FUNCTION_BLOCK L1_Merge2Cmd (* Basic Function Block Type *)
  (* Standard: 61499-2 *)
  (* Version 0.0, 2015-03-18, EQUEROL, UJI *)
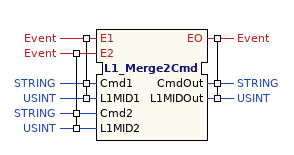
  EVENT_INPUT
    E1 WITH Cmd1, L1MID1; (* Event to merge 1 *)
    E2 WITH Cmd2, L1MID2; (* Event to merge 2 *)
  END_EVENT
  EVENT_OUTPUT
    EO WITH CmdOut, L1MIDOut; (* Initialization Confirm *)
  END_EVENT
  VAR_INPUT
    Cmd1 : STRING; (* Command with event 1 *)
    L1MID1 : USINT; (* Layer 1 multicast ID with 1 *)
    Cmd2 : STRING; (* Command with event 2 *)
    L1MID2 : USINT; (* Layer 1 multicast ID with 2 *)
  END_VAR
  VAR_OUTPUT
    CmdOut : STRING; (* Command out *)
    L1MIDOut : USINT; (* Layer 1 multicast ID *)
  END_VAR
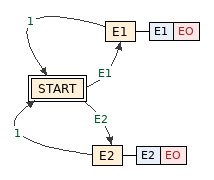
  EC_STATES
    START; (* Initial State *)
    E1 : E1 -> EO; (* Initialization *)
    E2 : E2 -> EO; (* Normal execution *)
  END_STATES
  EC_TRANSITIONS
    START TO E1 := E1;
    E1 TO START := 1;
    START TO E2 := E2;
    E2 TO START := 1;
  END_TRANSITIONS
  ALGORITHM E1 IN ST: (* Event 1 algo *)
CmdOut := Cmd1;
L1MIDOut := L1MID1;
  END_ALGORITHM
  ALGORITHM E2 IN ST: (* Event 2 algo *)
CmdOut := Cmd2;
L1MIDOut := L1MID2;
  END_ALGORITHM
END_FUNCTION_BLOCK
